Omron CX-Programmer project NewProject (CX-Programmer 9.73)

# PLC NewPLC1: CJ2M CPU32
I/O table (CPU CJ2M-CPU32): rack 0 slot 11 CJ2M-EIP21

## Program _1_feladat (cyclic task 0)
Local symbols
lm1 1.01 BOOL  ; léptetőmotor 1. tekercs
lm2 1.03 BOOL  ; léptetőmotor 2. tekercs
lm3 1.05 BOOL  ; léptetőmotor 3. tekercs
lm4 1.07 BOOL  ; léptetőmotor 4. tekercs
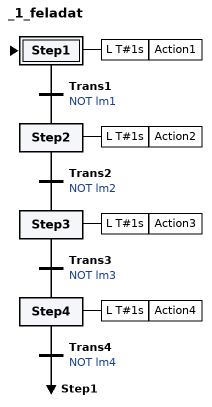
INITIAL_STEP Step1 :
Action1(L,T#1s) ;
END_STEP
TRANSITION Trans1 FROM Step1 TO Step2
 := NOT lm1;
END_TRANSITION
STEP Step2 :
Action2(L,T#1s) ;
END_STEP
TRANSITION Trans2 FROM Step2 TO Step3
 := NOT lm2;
END_TRANSITION
STEP Step3 :
Action3(L,T#1s) ;
END_STEP
TRANSITION Trans3 FROM Step3 TO Step4
 := NOT lm3;
END_TRANSITION
STEP Step4 :
Action4(L,T#1s) ;
END_STEP
TRANSITION Trans4 FROM Step4 TO Step1
 := NOT lm4;
END_TRANSITION

### Action Action1

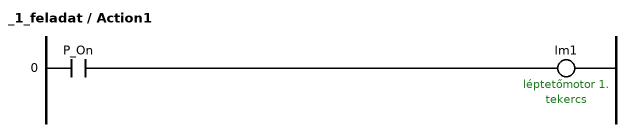
; rung 0
LD P_On
OUT lm1  ; léptetőmotor 1. tekercs

### Action Action2

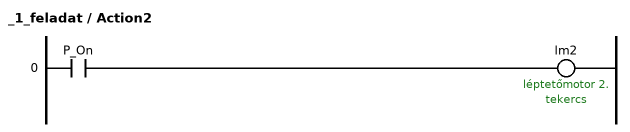
; rung 0
LD P_On
OUT lm2  ; léptetőmotor 2. tekercs

### Action Action3

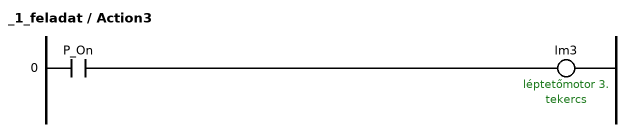
; rung 0
LD P_On
OUT lm3  ; léptetőmotor 3. tekercs

### Action Action4

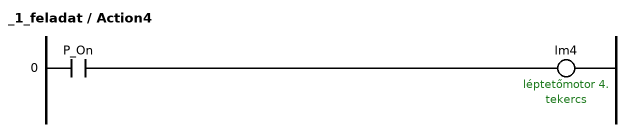
; rung 0
LD P_On
OUT lm4  ; léptetőmotor 4. tekercs

## Program _2_feladat (interrupt task -1)
Local symbols
lm1 1.01 BOOL  ; léptetőmotor 1. tekercs
lm2 1.03 BOOL  ; léptetőmotor 2. tekercs
lm3 1.05 BOOL  ; léptetőmotor 3. tekercs
lm4 1.07 BOOL  ; léptetőmotor 4. tekercs
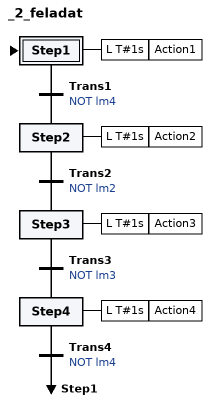
INITIAL_STEP Step1 :
Action1(L,T#1s) ;
END_STEP
TRANSITION Trans1 FROM Step1 TO Step2
 := NOT lm4;
END_TRANSITION
STEP Step2 :
Action2(L,T#1s) ;
END_STEP
TRANSITION Trans2 FROM Step2 TO Step3
 := NOT lm2;
END_TRANSITION
STEP Step3 :
Action3(L,T#1s) ;
END_STEP
TRANSITION Trans3 FROM Step3 TO Step4
 := NOT lm3;
END_TRANSITION
STEP Step4 :
Action4(L,T#1s) ;
END_STEP
TRANSITION Trans4 FROM Step4 TO Step1
 := NOT lm4;
END_TRANSITION

### Action Action1

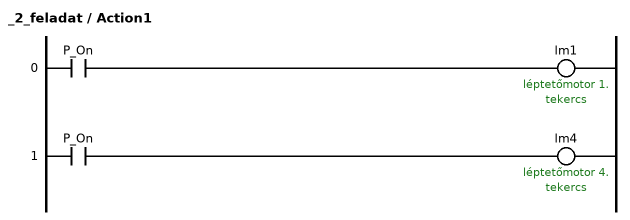
; rung 0
LD P_On
OUT lm1  ; léptetőmotor 1. tekercs
; rung 1
LD P_On
OUT lm4  ; léptetőmotor 4. tekercs

### Action Action2

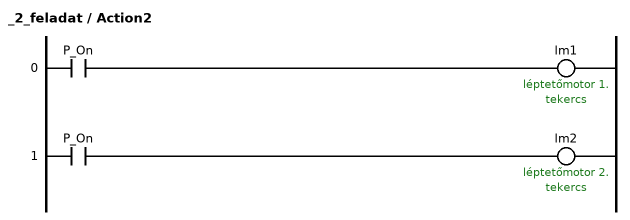
; rung 0
LD P_On
OUT lm1  ; léptetőmotor 1. tekercs
; rung 1
LD P_On
OUT lm2  ; léptetőmotor 2. tekercs

### Action Action3

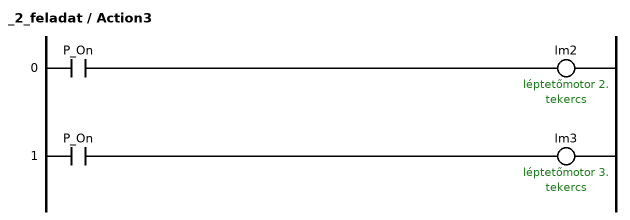
; rung 0
LD P_On
OUT lm2  ; léptetőmotor 2. tekercs
; rung 1
LD P_On
OUT lm3  ; léptetőmotor 3. tekercs

### Action Action4

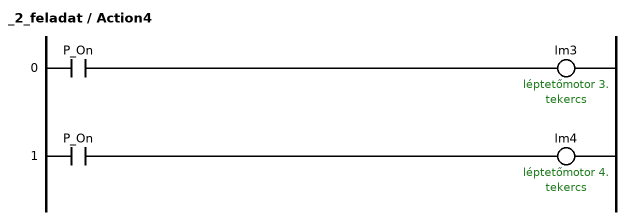
; rung 0
LD P_On
OUT lm3  ; léptetőmotor 3. tekercs
; rung 1
LD P_On
OUT lm4  ; léptetőmotor 4. tekercs

## Program _3_feladat (interrupt task -1)
Local symbols
lm1 1.01 BOOL  ; léptetőmotor 1. tekercs
lm2 1.03 BOOL  ; léptetőmotor 2. tekercs
lm3 1.05 BOOL  ; léptetőmotor 3. tekercs
lm4 1.07 BOOL  ; léptetőmotor 4. tekercs
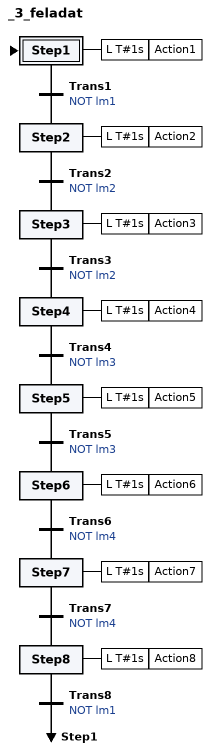
INITIAL_STEP Step1 :
Action1(L,T#1s) ;
END_STEP
TRANSITION Trans1 FROM Step1 TO Step2
 := NOT lm1;
END_TRANSITION
STEP Step2 :
Action2(L,T#1s) ;
END_STEP
TRANSITION Trans2 FROM Step2 TO Step3
 := NOT lm2;
END_TRANSITION
STEP Step3 :
Action3(L,T#1s) ;
END_STEP
TRANSITION Trans3 FROM Step3 TO Step4
 := NOT lm2;
END_TRANSITION
STEP Step4 :
Action4(L,T#1s) ;
END_STEP
TRANSITION Trans4 FROM Step4 TO Step5
 := NOT lm3;
END_TRANSITION
STEP Step5 :
Action5(L,T#1s) ;
END_STEP
TRANSITION Trans5 FROM Step5 TO Step6
 := NOT lm3;
END_TRANSITION
STEP Step6 :
Action6(L,T#1s) ;
END_STEP
TRANSITION Trans6 FROM Step6 TO Step7
 := NOT lm4;
END_TRANSITION
STEP Step7 :
Action7(L,T#1s) ;
END_STEP
TRANSITION Trans7 FROM Step7 TO Step8
 := NOT lm4;
END_TRANSITION
STEP Step8 :
Action8(L,T#1s) ;
END_STEP
TRANSITION Trans8 FROM Step8 TO Step1
 := NOT lm1;
END_TRANSITION

### Action Action1

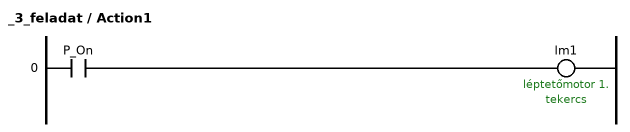
; rung 0
LD P_On
OUT lm1  ; léptetőmotor 1. tekercs

### Action Action2

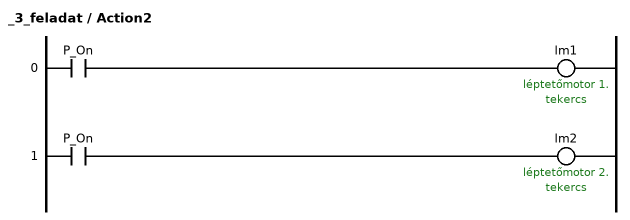
; rung 0
LD P_On
OUT lm1  ; léptetőmotor 1. tekercs
; rung 1
LD P_On
OUT lm2  ; léptetőmotor 2. tekercs

### Action Action3

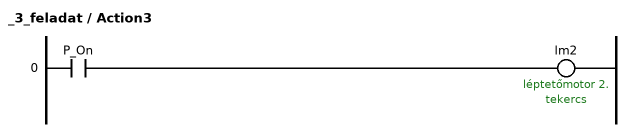
; rung 0
LD P_On
OUT lm2  ; léptetőmotor 2. tekercs

### Action Action4

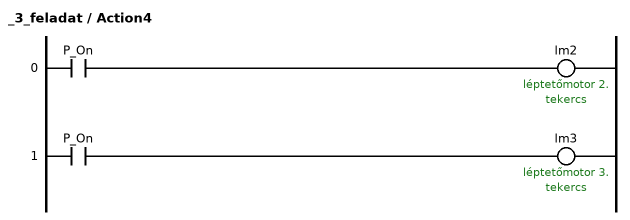
; rung 0
LD P_On
OUT lm2  ; léptetőmotor 2. tekercs
; rung 1
LD P_On
OUT lm3  ; léptetőmotor 3. tekercs

### Action Action5

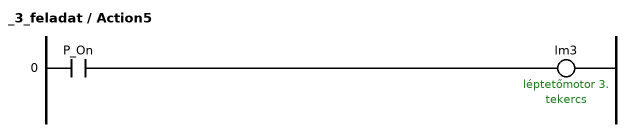
; rung 0
LD P_On
OUT lm3  ; léptetőmotor 3. tekercs

### Action Action6

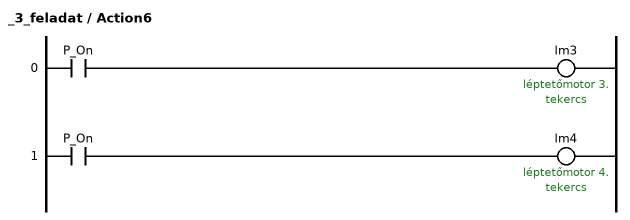
; rung 0
LD P_On
OUT lm3  ; léptetőmotor 3. tekercs
; rung 1
LD P_On
OUT lm4  ; léptetőmotor 4. tekercs

### Action Action7

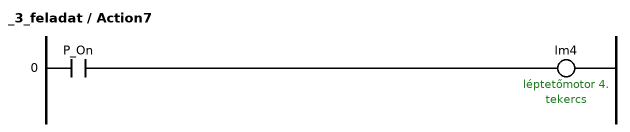
; rung 0
LD P_On
OUT lm4  ; léptetőmotor 4. tekercs

### Action Action8

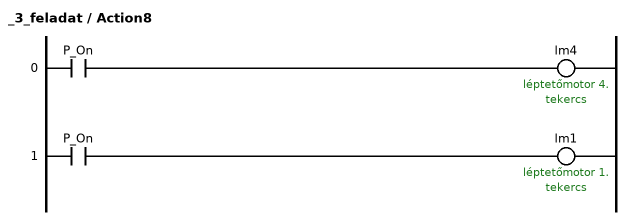
; rung 0
LD P_On
OUT lm4  ; léptetőmotor 4. tekercs
; rung 1
LD P_On
OUT lm1  ; léptetőmotor 1. tekercs

## Program _4_feladat (interrupt task -1)
Local symbols
i6 BOOL
ki1 1.00 BOOL
ki3 1.02 BOOL
ki4 1.03 BOOL
ki5 1.04 BOOL
ki6 1.05 BOOL
ki7 1.06 BOOL
ki8 1.07 BOOL
lm1 1.01 BOOL  ; léptetőmotor 1. tekercs
lm2 1.03 BOOL  ; léptetőmotor 2. tekercs
lm3 1.05 BOOL  ; léptetőmotor 3. tekercs
lm4 1.07 BOOL  ; léptetőmotor 4. tekercs
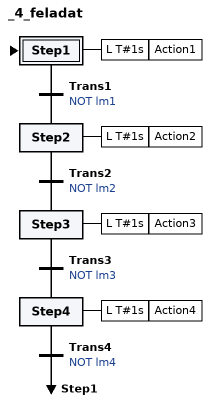
INITIAL_STEP Step1 :
Action1(L,T#1s) ;
END_STEP
TRANSITION Trans1 FROM Step1 TO Step2
 := NOT lm1;
END_TRANSITION
STEP Step2 :
Action2(L,T#1s) ;
END_STEP
TRANSITION Trans2 FROM Step2 TO Step3
 := NOT lm2;
END_TRANSITION
STEP Step3 :
Action3(L,T#1s) ;
END_STEP
TRANSITION Trans3 FROM Step3 TO Step4
 := NOT lm3;
END_TRANSITION
STEP Step4 :
Action4(L,T#1s) ;
END_STEP
TRANSITION Trans4 FROM Step4 TO Step1
 := NOT lm4;
END_TRANSITION

### Action Action1

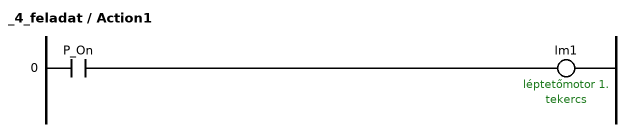
; rung 0
LD P_On
OUT lm1  ; léptetőmotor 1. tekercs

### Action Action2

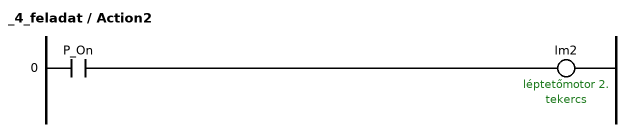
; rung 0
LD P_On
OUT lm2  ; léptetőmotor 2. tekercs

### Action Action3

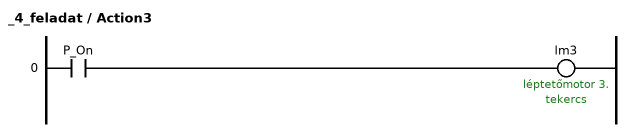
; rung 0
LD P_On
OUT lm3  ; léptetőmotor 3. tekercs

### Action Action4

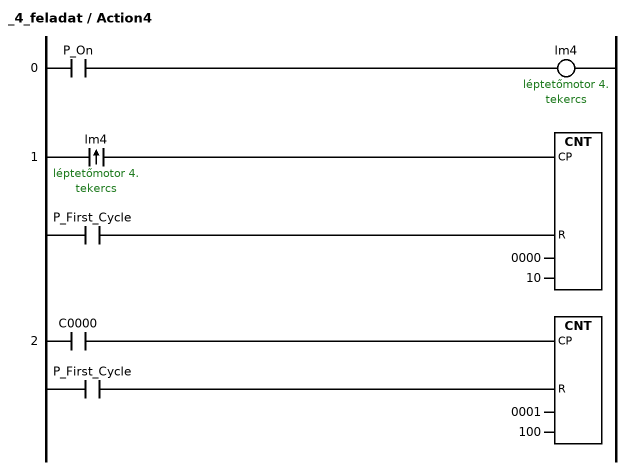
; rung 0
LD P_On
OUT lm4  ; léptetőmotor 4. tekercs
; rung 1
@LD lm4  ; léptetőmotor 4. tekercs
LD P_First_Cycle
CNT 0000 10
; rung 2
LD C0000
LD P_First_Cycle
CNT 0001 100

## Program _5_feladat (interrupt task -1)
Local symbols
ki1 1.00 BOOL
ki3 1.02 BOOL
ki5 1.04 BOOL
ki7 1.06 BOOL
lm1 1.01 BOOL  ; léptetőmotor 1. tekercs
lm2 1.03 BOOL  ; léptetőmotor 2. tekercs
lm3 1.05 BOOL  ; léptetőmotor 3. tekercs
lm4 1.07 BOOL  ; léptetőmotor 4. tekercs
